TYPE MoverStatus :
STRUCT
	isFrozen : BOOL;
	isLost : BOOL;
	isReadyForPositioning : BOOL;
	isActive : BOOL;
	hasDriveError : BOOL32;
	hasControllerError : BOOL32;
END_STRUCT
END_TYPE

(* stored: Version 1.1.0.1
   DUT MoverStatus: Id {f0f005da-3569-4cce-b174-391384937d02} *)
